TYPE ST_ITC_FunctionCommands :
(**************************************************************************************
 * 	Application		:	BoxControl Framework
 *	Revision		:	$Revision: 404529 $
 *	Revision date	:	$Date: 2018-04-23 08:21:38 +0200 (Mo., 23 Apr 2018) $
 *	Last changed by	:	$Author: b7bolm $
 *	URL				:	$URL: http://almscdc.swisslog.com/repo/SWPD/Development/BoxControlFramework/20_Release/trunk/01_Software/BCF/BCF/JumpStart/20_Product/10_App/12_E_Functions/10_Lib/10_Conv/01_DUTs/ST_ITC_FunctionCommands.TcDUT $
 *
 *	Purpose			:	Internal ITC function commands
 *
 * ------------------------------------------------------------------------------------
 *	Copyright Swisslog [IP AG], Switzerland. All rights reserved.
 * 
 * ------------------------------------------------------------------------------------
 *	
 * 	Revision History: 
 *
 * 	VERSION			DATE			INITIALS			DESCRIPTION
 *	0.1				01.01.2001		swl					Example
 *
 **************************************************************************************)
STRUCT
	StatusReport			: BOOL; // Command to send StatusReport 
	ControlReport			: BOOL; // Command to send ControlReport 
	NoErrorReport			: BOOL; // Command to send a 'no error' report
	ManualControlReport		: BOOL; // Command to send a manual control report
	ScannerInformationReport: BOOL; // Command to send a scanner information report
	ScannerNoReadReport		: BOOL; // Command to send a scanner no read report
END_STRUCT
END_TYPE

(* stored: Version 1.1.0.1, ProductVersion 3.1.4022.12
   DUT ST_ITC_FunctionCommands: Id {f37b77d1-4dbc-4af8-97f0-5c7a661c61ac} *)
